// TIA Portal V19 export
TYPE "LAF_typePlasticRollerEm6Parameters"
// stored: Access Published
   STRUCT
      cm1Vfd207 : "LAF_typeVfdParameters";
   END_STRUCT;
END_TYPE
